Staubli VAL3: check_table.pgx

program check_table(num& x_nInput[] (dimensions=2), bool& x_bResult)
  local num l_nElement
begin

  call util:rowSum(x_nInput, nResultRow)
  call util:colSum(x_nInput, nResultCol)
  x_bResult = false
  //check if ANY row or col is 0!

  for l_nElement = 0 to size(nResultRow)-1
    if nResultRow[l_nElement] == size(nResultRow)
      x_bResult = true
      return
    endIf
  endFor

  for l_nElement = 0 to size(nResultCol)-1
    if nResultCol[l_nElement] == size(nResultCol)
      x_bResult = true
      return
    endIf
  endFor


end
